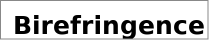
VISUALIZATION VISU_HMI_BIREFRINGENCE  // 209x40
    Label (10,10 199x30), "Birefringence"
END_VISUALIZATION

(* stored: Version 1.1.0.1, ProductVersion 3.1.4024.14
   Visu VISU_HMI_BIREFRINGENCE: Id {c93e8079-18e7-4190-ab63-1508a70dac3f} *)
